FUNCTION_BLOCK FB_TankController IMPLEMENTS I_TankController

VAR
	stTank :REFERENCE TO ST_Tank;
END_VAR

{warning 'add method implementation '}
METHOD ApplyCooling : BOOL
IF stTank.bAlarm THEN
	F_CoolTank(stTank);
END_IF
END_METHOD

{warning 'add method implementation '}
METHOD CheckSafety : BOOL
IF F_CheckAlarm( pTank := ADR(stTank) ) THEN
	stTank.bAlarm := TRUE;
END_IF
END_METHOD

METHOD FB_init : BOOL
VAR_INPUT
	bInitRetains : BOOL; // if TRUE, the retain variables are initialized (warm start / cold start)
	bInCopyCode : BOOL;  // if TRUE, the instance afterwards gets moved into the copy code (online change)
	_stTank : REFERENCE TO ST_TANK;
END_VAR
stTank REF= _stTank;
END_METHOD

METHOD StartController
VAR_INPUT
END_VAR
IF __ISVALIDREF(stTank) THEN
	CheckSafety();
	ApplyCooling();

	IF NOT stTank.bAlarm THEN
		stTank.fTemperature := stTank.fTemperature + 5;
	END_IF
END_IF
END_METHOD

END_FUNCTION_BLOCK

(* stored: Version 1.1.0.1, ProductVersion 3.1.4024.16
   POU FB_TankController: Id {bd5580ac-b1f3-4fa5-92f5-0a91a9517670}, SpecialFunc None
   Method ApplyCooling: Id {41f3f916-3681-4c60-b39a-5ab8cb364b13}
   Method CheckSafety: Id {dee3a59f-b24f-4a00-879d-a7220b0c9cf6}
   Method FB_init: Id {2140c440-63a9-4e57-8204-fd7f2509214b}
   Method StartController: Id {b987e19a-3d4a-4066-8261-4d90245bafb8} *)
